// TwinCAT 3 PLC project Lectures
// ProgramVersion: 3.1.4024.0
// libraries:
//   Tc2_Standard, * (Beckhoff Automation GmbH)
//   Tc2_System, * (Beckhoff Automation GmbH)
//   Tc3_Module, * (Beckhoff Automation GmbH)
// project tree:
//   DUTs/ Item.TcDUT (not stored), Location.TcDUT (not stored)
//   GVLs/ Automatic.TcGVL, IO.TcGVL
//   / PlcTask.TcTTO (not stored)
//   POUs/ AutomaticControl.TcPOU, CountPosition.TcPOU (not stored), Initialize.TcPOU, ManualControl.TcPOU, MAIN.TcPOU, MotorSelection.TcPOU, Recipe1.TcPOU, Recipe2.TcPOU, Safety.TcPOU
//   POUs/Lectures%27 programs/ p00_true_false.TcPOU (not stored), p01_sequential.TcPOU (not stored), p02_clock.TcPOU (not stored), p03_SR1.TcPOU (not stored), p04_latch.TcPOU (not stored), p05_posEdge.TcPOU (not stored), p06_frontDetection.TcPOU (not stored), p07_memoryCell.TcPOU (not stored), p08_counter.TcPOU (not stored), p09_timers.TcPOU (not stored), p10_directionalInterlock.TcPOU (not stored), p11_logicalFunction.TcPOU (not stored), p12_controlLight.TcPOU (not stored)
// real-time tasks:
//   TASK PlcTask1: cycle T#10ms, priority 21, ADS port 351
//   TASK PlcTask: cycle T#10ms, priority 20, ADS port 350
// I/O:
//   DEVICE Device 1 (EtherCAT), AmsNetId 172.31.192.1.2.1
//     Term 1 (EK1200) [EK1200-7000 EtherCAT Power supply (1,5A E-Bus)]
//       Term 2 (EL1859) [EL1859 8Ch. Dig. Input 24V, 3ms, 8Ch. Dig. Output 24V, 0.5A]
//       Term 3 (EL1859) [EL1859 8Ch. Dig. Input 24V, 3ms, 8Ch. Dig. Output 24V, 0.5A]
//       Term 4 (EL9011) [EL9011 End Terminal]
//   DEVICE Device 2 (NOV-DP-RAM) (disabled)
//   DEVICE Device 3 (CX7000), AmsNetId 172.31.192.1.4.1
//     Term 1 (CX7028) [CX7028-0000-0121]
//       modules: Module 1 (DIO_2x), Module 2 (Empty Module), Module 3 (DIO_2x), Module 4 (Empty Module), Module 5 (DI_2x), Module 6 (Empty Module), Module 7 (DI_2x), Module 8 (Empty Module)
// variable links:
//   Lectures/Lectures Instance <-> Device 1 (EtherCAT)/Term 1 (EK1200)/Term 2 (EL1859)
//     PlcTask Inputs/IO.EndExtensionSensor <-> Channel 3/Input
//     PlcTask Inputs/IO.EndGripSensor <-> Channel 7/Input
//     PlcTask Inputs/IO.EndLiftingSensor <-> Channel 5/Input
//     PlcTask Inputs/IO.EndRotationSensor <-> Channel 1/Input
//     PlcTask Inputs/IO.StepExtensionSwitch <-> Channel 4/Input
//     PlcTask Inputs/IO.StepGripSwitch <-> Channel 8/Input
//     PlcTask Inputs/IO.StepLiftingSwitch <-> Channel 6/Input
//     PlcTask Inputs/IO.StepRotatonSwitch <-> Channel 2/Input
//     PlcTask Outputs/IO.MotorExtension <-> Channel 12/Output
//     PlcTask Outputs/IO.MotorExtensionDirection <-> Channel 11/Output
//     PlcTask Outputs/IO.MotorGrip <-> Channel 16/Output
//     PlcTask Outputs/IO.MotorGripDirection <-> Channel 15/Output
//     PlcTask Outputs/IO.MotorLifting <-> Channel 14/Output
//     PlcTask Outputs/IO.MotorLiftingDirection <-> Channel 13/Output
//     PlcTask Outputs/IO.MotorRotation <-> Channel 10/Output
//     PlcTask Outputs/IO.MotorRotationDirection <-> Channel 9/Output
//   Lectures/Lectures Instance <-> Device 3 (CX7000)/Term 1 (CX7028)
//     PlcTask Inputs/IO.ButtonGreen <-> Module 3 (DIO_2x)/DIO_2x Input Channel 2/Input
//     PlcTask Inputs/IO.ButtonLowerLeft <-> Module 5 (DI_2x)/DI_2x Input Channel 1/Input
//     PlcTask Inputs/IO.ButtonLowerRight <-> Module 5 (DI_2x)/DI_2x Input Channel 2/Input
//     PlcTask Inputs/IO.ButtonRed <-> Module 1 (DIO_2x)/DIO_2x Input Channel 1/Input
//     PlcTask Inputs/IO.ButtonUpperLeft <-> Module 1 (DIO_2x)/DIO_2x Input Channel 2/Input
//     PlcTask Inputs/IO.ButtonUpperRight <-> Module 3 (DIO_2x)/DIO_2x Input Channel 1/Input
//     PlcTask Inputs/IO.Switch <-> Module 7 (DI_2x)/DI_2x Input Channel 1/Input
//     PlcTask Outputs/IO.LEDBlueLower <-> Module 3 (DIO_2x)/DIO_2x Output Channel 2/Output
//     PlcTask Outputs/IO.LEDBlueUpper <-> Module 1 (DIO_2x)/DIO_2x Output Channel 2/Output
//     PlcTask Outputs/IO.LEDGreen <-> Module 3 (DIO_2x)/DIO_2x Output Channel 1/Output
//     PlcTask Outputs/IO.LEDRed <-> Module 1 (DIO_2x)/DIO_2x Output Channel 1/Output

// ---- GVLs/Automatic.TcGVL
{attribute 'qualified_only'}
VAR_GLOBAL
	SwitchedON: BOOL;
	CurrentLocation: Location;
	CurrentSelection: INT;
	//MotorRot: Motors;
	//MotorLif: Motors;
	//MotorExt: Motors;
	//MotorGri: Motors;
	
	RotationPositionAuto: INT;
	RotationPositionCurrent: INT;
	RotationMovement: BOOL;
	
	LiftingPositionAuto: INT;
	LiftingPositionCurrent: INT;
	LiftingMovement: BOOL;
	
	ExtensionPositionAuto: INT;
	ExtensionPositionCurrent: INT;
	ExtensionMovement: BOOL;
	
	GripPositionAuto: INT;
	GripPositionCurrent: INT;
	GripMovement: BOOL;
END_VAR

// ---- GVLs/IO.TcGVL
{attribute 'qualified_only'}
VAR_GLOBAL
	ButtonRed AT %I*: BOOL;
	ButtonUpperRight AT %I*: BOOL;
	ButtonLowerLeft AT %I*: BOOL;
	Switch AT %I*: BOOL;
	LEDRed AT %Q*: BOOL;
	LEDGreen AT %Q*: BOOL;
	ButtonUpperLeft AT %I*: BOOL;
	ButtonGreen AT %I*: BOOL;
	ButtonLowerRight AT %I*: BOOL;
	LEDBlueUpper AT %Q*: BOOL;
	LEDBlueLower AT %Q*: BOOL;
	
	EndRotationSensor AT %I*: BOOL;
	StepRotatonSwitch AT %I*: BOOL;
	EndExtensionSensor AT %I*: BOOL;
	StepExtensionSwitch AT %I*: BOOL;
	EndLiftingSensor AT %I*: BOOL;
	StepLiftingSwitch AT %I*: BOOL;
	EndGripSensor AT %I*: BOOL;
	StepGripSwitch AT %I*: BOOL;
	MotorRotationDirection AT %Q*: BOOL;
	MotorRotation AT %Q*: BOOL;
	MotorExtensionDirection AT %Q*: BOOL;
	MotorExtension AT %Q*: BOOL;
	MotorLiftingDirection AT %Q*: BOOL;
	MotorLifting AT %Q*: BOOL;
	MotorGripDirection AT %Q*: BOOL;
	MotorGrip AT %Q*: BOOL;
	Initialized: BOOL;
	MotorDirection: INT;
	SwitchedToAutomatic: BOOL;
END_VAR

// ---- POUs/AutomaticControl.TcPOU
FUNCTION_BLOCK PUBLIC AutomaticControl
VAR_INPUT
	Switch: BOOL;
END_VAR
VAR
	ExecutingRecipe1: BOOL := FALSE;
	ExecutingRecipe2: BOOL := FALSE;
	SwitchedManualAuto: BOOL := FALSE;
	initialized: BOOL := FALSE;
	State: INT := 0;
END_VAR
VAR_OUTPUT
	Output: BOOL;
END_VAR

// Initially go to position (0,0,0,0) and initialize motors
IF NOT IO.Initialized THEN
	Initialize();
ELSE
	//Safety();	// to stop when out of range
	
	// COUNTING (POSITION):
	CountPosition();	// FOR MANUAL MODE
	
	// RESET THE POSITION:
	(*IF (Automatic.RotationPositionAuto - Automatic.RotationPositionCurrent > 20 OR Automatic.RotationPositionAuto - Automatic.RotationPositionCurrent > 20) AND IO.SwitchedToAutomatic THEN
		IF Automatic.RotationPositionAuto - Automatic.RotationPositionCurrent > 20 THEN
			IO.MotorRotationDirection := 0;
		ELSE
			IO.MotorRotationDirection := 1;
		END_IF
		IO.MotorRotation := 1;
	ELSE 
		IO.MotorRotation := 0;
		IO.SwitchedToAutomatic := 0;
	END_IF*)
	(*IF Automatic.ExtensionPositionAuto <> Automatic.ExtensionPositionCurrent AND NOT IO.Switch THEN
		IF Automatic.ExtensionPositionAuto - Automatic.ExtensionPositionCurrent > 0 THEN
			IO.MotorExtensionDirection := 0;
		ELSE
			IO.MotorExtensionDirection := 1;
		END_IF
		IO.MotorExtension := 1;
	ELSE 
		IF NOT IO.Switch THEN
			IO.MotorExtension := 0;
		END_IF
	END_IF*)
	
	
	
	// RECIPES (recipe is sequence of moves to execute the task):
	IF ExecutingRecipe1 OR IO.ButtonUpperLeft THEN
		ExecutingRecipe1 := TRUE;
		Recipe1();
		ExecutingRecipe1 := NOT Recipe1.Ended;
	ELSIF NOT ExecutingRecipe1 AND (IO.ButtonUpperRight OR ExecutingRecipe2) THEN
		ExecutingRecipe2 := TRUE;
		Recipe2();
		ExecutingRecipe2 := NOT Recipe2.Ended;
	END_IF
	
END_IF

// for debugging purposes:
IF IO.ButtonRed THEN
	IO.Initialized := FALSE;
END_IF

RETURN;

END_FUNCTION_BLOCK

// ---- POUs/Initialize.TcPOU
PROGRAM Initialize
VAR
END_VAR

// go to the initial position (0,0,0,0)
IF IO.EndRotationSensor THEN
	IO.MotorRotation := 0;
	IO.MotorRotationDirection := 0;
ELSE 
	IO.MotorRotationDirection := 1;
	IO.MotorRotation := 1;
END_IF

IF IO.EndLiftingSensor THEN
	IO.MotorLifting := 0;
	IO.MotorLiftingDirection := 0;
ELSE 
	IO.MotorLiftingDirection := 1;
	IO.MotorLifting := 1;
END_IF

IF IO.EndExtensionSensor THEN
	IO.MotorExtension := 0;
	IO.MotorExtensionDirection := 0;
ELSE 
	IO.MotorExtensionDirection := 1;
	IO.MotorExtension := 1;
END_IF

IF IO.EndGripSensor THEN
	IO.MotorGrip := 0;
	IO.MotorGripDirection := 0;
ELSE 
	IO.MotorGripDirection := 1;
	IO.MotorGrip := 1;
END_IF
	
IF IO.EndRotationSensor AND IO.EndLiftingSensor AND IO.EndExtensionSensor AND IO.EndGripSensor THEN
	IO.Initialized := TRUE;
END_IF

END_PROGRAM

// ---- POUs/Recipe1.TcPOU
PROGRAM Recipe1
VAR
	State: INT := 0;
END_VAR

IF State = 24 AND IO.ButtonGreen THEN	// reinitialize and run the recipe again on green button press
	IO.Initialized := 0;
	State := 0;
END_IF

IF IO.Initialized AND NOT IO.Switch THEN
	
	// delay...
	// vrni se v stanje ob preklopu...
	// daj v funkcije in kliči, namesto PRG...
	// Recipe2...
	
	// WOOD:
	IF State = 0 THEN
		IF Automatic.LiftingPositionAuto < 50 THEN
			IO.MotorLiftingDirection := 0;
			IO.MotorLifting := 1;
			Automatic.LiftingPositionAuto := Automatic.LiftingPositionAuto + 1;
			Automatic.LiftingPositionCurrent := Automatic.LiftingPositionCurrent + 1;
		ELSE
			State := 1;
			IO.MotorLifting := 0;
		END_IF
	ELSIF State = 1 THEN
		IF Automatic.ExtensionPositionAuto < 388 THEN
			IO.MotorExtensionDirection := 0;
			IO.MotorExtension := 1;
			Automatic.ExtensionPositionAuto := Automatic.ExtensionPositionAuto + 1;
			Automatic.ExtensionPositionCurrent := Automatic.ExtensionPositionCurrent + 1;
		ELSE
			State := 2;
			IO.MotorExtension := 0;
		END_IF
	ELSIF State = 2 THEN
		IF Automatic.GripPositionAuto < 160 THEN
			IO.MotorGripDirection := 0;
			IO.MotorGrip := 1;
			Automatic.GripPositionAuto := Automatic.GripPositionAuto + 1;
			Automatic.GripPositionCurrent := Automatic.GripPositionCurrent + 1;
		ELSE
			State := 3;
			IO.MotorGrip := 0;
		END_IF
	ELSIF State = 3 THEN
		IF NOT IO.EndLiftingSensor THEN
			IO.MotorLiftingDirection := 0;
			IO.MotorLifting := 1;
			Automatic.LiftingPositionAuto := Automatic.LiftingPositionAuto - 1;
			Automatic.LiftingPositionCurrent := Automatic.LiftingPositionCurrent - 1;
		ELSE
			State := 4;
			IO.MotorLifting := 0;
		END_IF
	ELSIF State = 4 THEN
		IF Automatic.RotationPositionAuto < 300 THEN
			IO.MotorRotationDirection := 0;
			IO.MotorRotation := 1;
			Automatic.RotationPositionAuto := Automatic.RotationPositionAuto + 1;
			Automatic.RotationPositionCurrent := Automatic.RotationPositionCurrent + 1;
		ELSE
			State := 5;
			IO.MotorRotation := 0;
		END_IF
	ELSIF State = 5 THEN
		IF NOT IO.EndExtensionSensor THEN	// it drops wood in the nearest bin
			IO.MotorExtensionDirection := 1;
			IO.MotorExtension := 1;
			Automatic.ExtensionPositionAuto := Automatic.ExtensionPositionAuto - 1;
			Automatic.ExtensionPositionCurrent := Automatic.ExtensionPositionCurrent - 1;
		ELSE
			State := 6;
			IO.MotorExtension := 0;
		END_IF
	ELSIF State = 6 THEN
		IF NOT IO.EndGripSensor THEN
			IO.MotorGripDirection := 1;
			IO.MotorGrip := 1;
			Automatic.GripPositionAuto := Automatic.GripPositionAuto - 1;
			Automatic.GripPositionCurrent := Automatic.GripPositionCurrent - 1;
		ELSE
			State := 7;
			IO.MotorGrip := 0;
		END_IF
	ELSIF State = 7 THEN
		IF NOT IO.EndRotationSensor THEN
			IO.MotorRotationDirection := 1;
			IO.MotorRotation := 1;
			Automatic.RotationPositionAuto := Automatic.RotationPositionAuto - 1;
			Automatic.RotationPositionCurrent := Automatic.RotationPositionCurrent - 1;
		ELSE
			State := 8;
			IO.MotorRotation := 0;
		END_IF
	END_IF
	
	// PLASTICS:
	IF State = 8 THEN
		IF Automatic.LiftingPositionAuto < 250 THEN
			IO.MotorLiftingDirection := 0;
			IO.MotorLifting := 1;
			Automatic.LiftingPositionAuto := Automatic.LiftingPositionAuto + 1;
			Automatic.LiftingPositionCurrent := Automatic.LiftingPositionCurrent + 1;
		ELSE
			State := 9;
			IO.MotorLifting := 0;
		END_IF
	ELSIF State = 9 THEN
		IF Automatic.ExtensionPositionAuto < 388 THEN
			IO.MotorExtensionDirection := 0;
			IO.MotorExtension := 1;
			Automatic.ExtensionPositionAuto := Automatic.ExtensionPositionAuto + 1;
			Automatic.ExtensionPositionCurrent := Automatic.ExtensionPositionCurrent + 1;
		ELSE
			State := 10;
			IO.MotorExtension := 0;
		END_IF
	ELSIF State = 10 THEN
		IF Automatic.GripPositionAuto < 160 THEN
			IO.MotorGripDirection := 0;
			IO.MotorGrip := 1;
			Automatic.GripPositionAuto := Automatic.GripPositionAuto + 1;
			Automatic.GripPositionCurrent := Automatic.GripPositionCurrent + 1;
		ELSE
			State := 11;
			IO.MotorGrip := 0;
		END_IF
	ELSIF State = 11 THEN
		IF NOT IO.EndLiftingSensor THEN
			IO.MotorLiftingDirection := 1;
			IO.MotorLifting := 1;
			Automatic.LiftingPositionAuto := Automatic.LiftingPositionAuto - 1;
			Automatic.LiftingPositionCurrent := Automatic.LiftingPositionCurrent - 1;
		ELSE
			State := 12;
			IO.MotorLifting := 0;
		END_IF
	ELSIF State = 12 THEN
		IF Automatic.RotationPositionAuto < 300 THEN
			IO.MotorRotationDirection := 0;
			IO.MotorRotation := 1;
			Automatic.RotationPositionAuto := Automatic.RotationPositionAuto + 1;
			Automatic.RotationPositionCurrent := Automatic.RotationPositionCurrent + 1;
		ELSE
			State := 13;
			IO.MotorRotation := 0;
		END_IF
	ELSIF State = 13 THEN
		IF Automatic.ExtensionPositionAuto > 300 THEN	// it drops plastics into second nearest bin
			IO.MotorExtensionDirection := 1;
			IO.MotorExtension := 1;
			Automatic.ExtensionPositionAuto := Automatic.ExtensionPositionAuto - 1;
			Automatic.ExtensionPositionCurrent := Automatic.ExtensionPositionCurrent - 1;
		ELSE
			State := 14;
			IO.MotorExtensionDirection := 0;
			IO.MotorExtension := 0;
		END_IF
	ELSIF State = 14 THEN
		IF NOT IO.EndGripSensor THEN
			IO.MotorGripDirection := 1;
			IO.MotorGrip := 1;
			Automatic.GripPositionAuto := Automatic.GripPositionAuto - 1;
			Automatic.GripPositionCurrent := Automatic.GripPositionCurrent - 1;
		ELSE
			State := 15;
			IO.MotorGrip := 0;
		END_IF
	ELSIF State = 15 THEN
		IF NOT IO.EndRotationSensor THEN
			IO.MotorRotationDirection := 1;
			IO.MotorRotation := 1;
			Automatic.RotationPositionAuto := Automatic.RotationPositionAuto - 1;
			Automatic.RotationPositionCurrent := Automatic.RotationPositionCurrent - 1;
		ELSE
			State := 16;
			IO.MotorRotation := 0;
		END_IF
	END_IF
	
	// METAL:
	IF State = 16 THEN
		IF Automatic.LiftingPositionAuto < 400 THEN
			IO.MotorLiftingDirection := 0;
			IO.MotorLifting := 1;
			Automatic.LiftingPositionAuto := Automatic.LiftingPositionAuto + 1;
			Automatic.LiftingPositionCurrent := Automatic.LiftingPositionCurrent + 1;
		ELSE
			State := 17;
			IO.MotorLifting := 0;
		END_IF
	ELSIF State = 17 THEN
		IF Automatic.ExtensionPositionAuto < 388 THEN
			IO.MotorExtensionDirection := 0;
			IO.MotorExtension := 1;
			Automatic.ExtensionPositionAuto := Automatic.ExtensionPositionAuto + 1;
			Automatic.ExtensionPositionCurrent := Automatic.ExtensionPositionCurrent + 1;
		ELSE
			State := 18;
			IO.MotorExtension := 0;
		END_IF
	ELSIF State = 18 THEN
		IF Automatic.GripPositionAuto < 160 THEN
			IO.MotorGripDirection := 0;
			IO.MotorGrip := 1;
			Automatic.GripPositionAuto := Automatic.GripPositionAuto + 1;
			Automatic.GripPositionCurrent := Automatic.GripPositionCurrent + 1;
		ELSE
			State := 19;
			IO.MotorGrip := 0;
		END_IF
	ELSIF State = 19 THEN
		IF NOT IO.EndLiftingSensor THEN
			IO.MotorLiftingDirection := 1;
			IO.MotorLifting := 1;
			Automatic.LiftingPositionAuto := Automatic.LiftingPositionAuto - 1;
			Automatic.LiftingPositionCurrent := Automatic.LiftingPositionCurrent - 1;
		ELSE
			State := 20;
			IO.MotorLifting := 0;
		END_IF
	ELSIF State = 20 THEN
		IF Automatic.RotationPositionAuto < 300 THEN
			IO.MotorRotationDirection := 0;
			IO.MotorRotation := 1;
			Automatic.RotationPositionAuto := Automatic.RotationPositionAuto + 1;
			Automatic.RotationPositionCurrent := Automatic.RotationPositionCurrent + 1;
		ELSE
			State := 21;
			IO.MotorRotation := 0;
		END_IF
	ELSIF State = 21 THEN
		IF Automatic.ExtensionPositionAuto > 500 THEN	// it drops metal into farthest bin
			IO.MotorExtensionDirection := 1;
			IO.MotorExtension := 1;
			Automatic.ExtensionPositionAuto := Automatic.ExtensionPositionAuto - 1;
			Automatic.ExtensionPositionCurrent := Automatic.ExtensionPositionCurrent - 1;
		ELSE
			State := 22;
			IO.MotorExtension := 0;
		END_IF
	ELSIF State = 22 THEN
		IF NOT IO.EndGripSensor THEN
			IO.MotorGripDirection := 1;
			IO.MotorGrip := 1;
			Automatic.GripPositionAuto := Automatic.GripPositionAuto - 1;
			Automatic.GripPositionCurrent := Automatic.GripPositionCurrent - 1;
		ELSE
			State := 23;
			IO.MotorGrip := 0;
		END_IF
	ELSIF State = 23 THEN
		IF NOT IO.EndRotationSensor THEN
			IO.MotorRotationDirection := 1;
			IO.MotorRotation := 1;
			Automatic.RotationPositionAuto := Automatic.RotationPositionAuto - 1;
			Automatic.RotationPositionCurrent := Automatic.RotationPositionCurrent - 1;
		ELSE
			State := 24;
			IO.MotorRotation := 0;
		END_IF
	END_IF
END_IF

END_PROGRAM

// ---- POUs/Recipe2.TcPOU
PROGRAM Recipe2
VAR
	State: INT := 8;
	Ended: BOOL := FALSE;
END_VAR

IF State = 24 AND IO.ButtonGreen THEN	// reinitialize and run the recipe again on green button press
	IO.Initialized := 0;
	State := 0;
END_IF

IF IO.Initialized AND NOT IO.Switch THEN
	
	// WOOD:
	IF State = 0 THEN
		IF Automatic.LiftingPositionAuto < 50 THEN
			IO.MotorLiftingDirection := 0;
			IO.MotorLifting := 1;
			Automatic.LiftingPositionAuto := Automatic.LiftingPositionAuto + 1;
			Automatic.LiftingPositionCurrent := Automatic.LiftingPositionCurrent + 1;
		ELSE
			State := 1;
			IO.MotorLifting := 0;
		END_IF
	ELSIF State = 1 THEN
		IF Automatic.ExtensionPositionAuto < 388 THEN
			IO.MotorExtensionDirection := 0;
			IO.MotorExtension := 1;
			Automatic.ExtensionPositionAuto := Automatic.ExtensionPositionAuto + 1;
			Automatic.ExtensionPositionCurrent := Automatic.ExtensionPositionCurrent + 1;
		ELSE
			State := 2;
			IO.MotorExtension := 0;
		END_IF
	ELSIF State = 2 THEN
		IF Automatic.GripPositionAuto < 160 THEN
			IO.MotorGripDirection := 0;
			IO.MotorGrip := 1;
			Automatic.GripPositionAuto := Automatic.GripPositionAuto + 1;
			Automatic.GripPositionCurrent := Automatic.GripPositionCurrent + 1;
		ELSE
			State := 3;
			IO.MotorGrip := 0;
		END_IF
	ELSIF State = 3 THEN
		IF NOT IO.EndLiftingSensor THEN
			IO.MotorLiftingDirection := 1;
			IO.MotorLifting := 1;
			Automatic.LiftingPositionAuto := Automatic.LiftingPositionAuto - 1;
			Automatic.LiftingPositionCurrent := Automatic.LiftingPositionCurrent - 1;
		ELSE
			State := 4;
			IO.MotorLifting := 0;
		END_IF
	ELSIF State = 4 THEN
		IF Automatic.RotationPositionAuto < 300 THEN
			IO.MotorRotationDirection := 0;
			IO.MotorRotation := 1;
			Automatic.RotationPositionAuto := Automatic.RotationPositionAuto + 1;
			Automatic.RotationPositionCurrent := Automatic.RotationPositionCurrent + 1;
		ELSE
			State := 5;
			IO.MotorRotation := 0;
		END_IF
	ELSIF State = 5 THEN
		IF NOT IO.EndExtensionSensor THEN	// it drops wood in the nearest bin
			IO.MotorExtensionDirection := 1;
			IO.MotorExtension := 1;
			Automatic.ExtensionPositionAuto := Automatic.ExtensionPositionAuto - 1;
			Automatic.ExtensionPositionCurrent := Automatic.ExtensionPositionCurrent - 1;
		ELSE
			State := 6;
			IO.MotorExtension := 0;
		END_IF
	ELSIF State = 6 THEN
		IF NOT IO.EndGripSensor THEN
			IO.MotorGripDirection := 1;
			IO.MotorGrip := 1;
			Automatic.GripPositionAuto := Automatic.GripPositionAuto - 1;
			Automatic.GripPositionCurrent := Automatic.GripPositionCurrent - 1;
		ELSE
			State := 7;
			IO.MotorGrip := 0;
		END_IF
	ELSIF State = 7 THEN
		IF NOT IO.EndRotationSensor THEN
			IO.MotorRotationDirection := 1;
			IO.MotorRotation := 1;
			Automatic.RotationPositionAuto := Automatic.RotationPositionAuto - 1;
			Automatic.RotationPositionCurrent := Automatic.RotationPositionCurrent - 1;
		ELSE
			State := 8;
			IO.MotorRotation := 0;
		END_IF
	END_IF
	
	// PLASTICS:
	IF State = 8 THEN
		IF Automatic.LiftingPositionAuto < 250 THEN
			IO.MotorLiftingDirection := 0;
			IO.MotorLifting := 1;
			Automatic.LiftingPositionAuto := Automatic.LiftingPositionAuto + 1;
			Automatic.LiftingPositionCurrent := Automatic.LiftingPositionCurrent + 1;
		ELSE
			State := 9;
			IO.MotorLifting := 0;
		END_IF
	ELSIF State = 9 THEN
		IF Automatic.ExtensionPositionAuto < 388 THEN
			IO.MotorExtensionDirection := 0;
			IO.MotorExtension := 1;
			Automatic.ExtensionPositionAuto := Automatic.ExtensionPositionAuto + 1;
			Automatic.ExtensionPositionCurrent := Automatic.ExtensionPositionCurrent + 1;
		ELSE
			State := 10;
			IO.MotorExtension := 0;
		END_IF
	ELSIF State = 10 THEN
		IF Automatic.GripPositionAuto < 160 THEN
			IO.MotorGripDirection := 0;
			IO.MotorGrip := 1;
			Automatic.GripPositionAuto := Automatic.GripPositionAuto + 1;
			Automatic.GripPositionCurrent := Automatic.GripPositionCurrent + 1;
		ELSE
			State := 11;
			IO.MotorGrip := 0;
		END_IF
	ELSIF State = 11 THEN
		IF NOT IO.EndLiftingSensor THEN
			IO.MotorLiftingDirection := 1;
			IO.MotorLifting := 1;
			Automatic.LiftingPositionAuto := Automatic.LiftingPositionAuto - 1;
			Automatic.LiftingPositionCurrent := Automatic.LiftingPositionCurrent - 1;
		ELSE
			State := 12;
			IO.MotorLifting := 0;
		END_IF
	ELSIF State = 12 THEN
		IF Automatic.RotationPositionAuto < 300 THEN
			IO.MotorRotationDirection := 0;
			IO.MotorRotation := 1;
			Automatic.RotationPositionAuto := Automatic.RotationPositionAuto + 1;
			Automatic.RotationPositionCurrent := Automatic.RotationPositionCurrent + 1;
		ELSE
			State := 13;
			IO.MotorRotation := 0;
		END_IF
	ELSIF State = 13 THEN
		IF Automatic.ExtensionPositionAuto > 300 THEN	// it drops plastics into second nearest bin
			IO.MotorExtensionDirection := 1;
			IO.MotorExtension := 1;
			Automatic.ExtensionPositionAuto := Automatic.ExtensionPositionAuto - 1;
			Automatic.ExtensionPositionCurrent := Automatic.ExtensionPositionCurrent - 1;
		ELSE
			State := 14;
			IO.MotorExtensionDirection := 0;
			IO.MotorExtension := 0;
		END_IF
	ELSIF State = 14 THEN
		IF NOT IO.EndGripSensor THEN
			IO.MotorGripDirection := 1;
			IO.MotorGrip := 1;
			Automatic.GripPositionAuto := Automatic.GripPositionAuto - 1;
			Automatic.GripPositionCurrent := Automatic.GripPositionCurrent - 1;
		ELSE
			State := 15;
			IO.MotorGrip := 0;
		END_IF
	ELSIF State = 15 THEN
		IF NOT IO.EndRotationSensor THEN
			IO.MotorRotationDirection := 1;
			IO.MotorRotation := 1;
			Automatic.RotationPositionAuto := Automatic.RotationPositionAuto - 1;
			Automatic.RotationPositionCurrent := Automatic.RotationPositionCurrent - 1;
		ELSE
			State := 16;
			IO.MotorRotation := 0;
		END_IF
	END_IF
	
	// METAL:
	IF State = 16 THEN
		IF Automatic.LiftingPositionAuto < 400 THEN
			IO.MotorLiftingDirection := 0;
			IO.MotorLifting := 1;
			Automatic.LiftingPositionAuto := Automatic.LiftingPositionAuto + 1;
			Automatic.LiftingPositionCurrent := Automatic.LiftingPositionCurrent + 1;
		ELSE
			State := 17;
			IO.MotorLifting := 0;
		END_IF
	ELSIF State = 17 THEN
		IF Automatic.ExtensionPositionAuto < 388 THEN
			IO.MotorExtensionDirection := 0;
			IO.MotorExtension := 1;
			Automatic.ExtensionPositionAuto := Automatic.ExtensionPositionAuto + 1;
			Automatic.ExtensionPositionCurrent := Automatic.ExtensionPositionCurrent + 1;
		ELSE
			State := 18;
			IO.MotorExtension := 0;
		END_IF
	ELSIF State = 18 THEN
		IF Automatic.GripPositionAuto < 160 THEN
			IO.MotorGripDirection := 0;
			IO.MotorGrip := 1;
			Automatic.GripPositionAuto := Automatic.GripPositionAuto + 1;
			Automatic.GripPositionCurrent := Automatic.GripPositionCurrent + 1;
		ELSE
			State := 19;
			IO.MotorGrip := 0;
		END_IF
	ELSIF State = 19 THEN
		IF NOT IO.EndLiftingSensor THEN
			IO.MotorLiftingDirection := 1;
			IO.MotorLifting := 1;
			Automatic.LiftingPositionAuto := Automatic.LiftingPositionAuto - 1;
			Automatic.LiftingPositionCurrent := Automatic.LiftingPositionCurrent - 1;
		ELSE
			State := 20;
			IO.MotorLifting := 0;
		END_IF
	ELSIF State = 20 THEN
		IF Automatic.RotationPositionAuto < 300 THEN
			IO.MotorRotationDirection := 0;
			IO.MotorRotation := 1;
			Automatic.RotationPositionAuto := Automatic.RotationPositionAuto + 1;
			Automatic.RotationPositionCurrent := Automatic.RotationPositionCurrent + 1;
		ELSE
			State := 21;
			IO.MotorRotation := 0;
		END_IF
	ELSIF State = 21 THEN
		IF Automatic.ExtensionPositionAuto > 500 THEN	// it drops metal into farthest bin
			IO.MotorExtensionDirection := 1;
			IO.MotorExtension := 1;
			Automatic.ExtensionPositionAuto := Automatic.ExtensionPositionAuto - 1;
			Automatic.ExtensionPositionCurrent := Automatic.ExtensionPositionCurrent - 1;
		ELSE
			State := 22;
			IO.MotorExtension := 0;
		END_IF
	ELSIF State = 22 THEN
		IF NOT IO.EndGripSensor THEN
			IO.MotorGripDirection := 1;
			IO.MotorGrip := 1;
			Automatic.GripPositionAuto := Automatic.GripPositionAuto - 1;
			Automatic.GripPositionCurrent := Automatic.GripPositionCurrent - 1;
		ELSE
			State := 23;
			IO.MotorGrip := 0;
		END_IF
	ELSIF State = 23 THEN
		IF NOT IO.EndRotationSensor THEN
			IO.MotorRotationDirection := 1;
			IO.MotorRotation := 1;
			Automatic.RotationPositionAuto := Automatic.RotationPositionAuto - 1;
			Automatic.RotationPositionCurrent := Automatic.RotationPositionCurrent - 1;
		ELSE
			State := 24;
			IO.MotorRotation := 0;
		END_IF
	ELSIF State = 24 THEN
		State := 8;
		Ended := TRUE;
	END_IF
END_IF

END_PROGRAM

// ---- POUs/ManualControl.TcPOU
FUNCTION_BLOCK PUBLIC ManualControl
VAR_INPUT
	Switch: BOOL;
END_VAR
VAR
	ManualControl: BOOL;
	TimeForInterlockDelay: TIME := T#0.05S;
	ManualMode: BOOL;
	MotorSelection_1: MotorSelection;
	SelectedMotor: INT;
	temp: TIME;
	LowerLeftInterlock: TOF;
	LowerLeft: BOOL;
	LowerRightInterlock: TOF;
	LowerRight: BOOL;
END_VAR
VAR_OUTPUT
	Output: BOOL;
END_VAR
VAR // added by the converter: edge detectors and wires of the graphical bodies
    _w1, _w2, _w3, _w4, _w5 : BOOL;
END_VAR

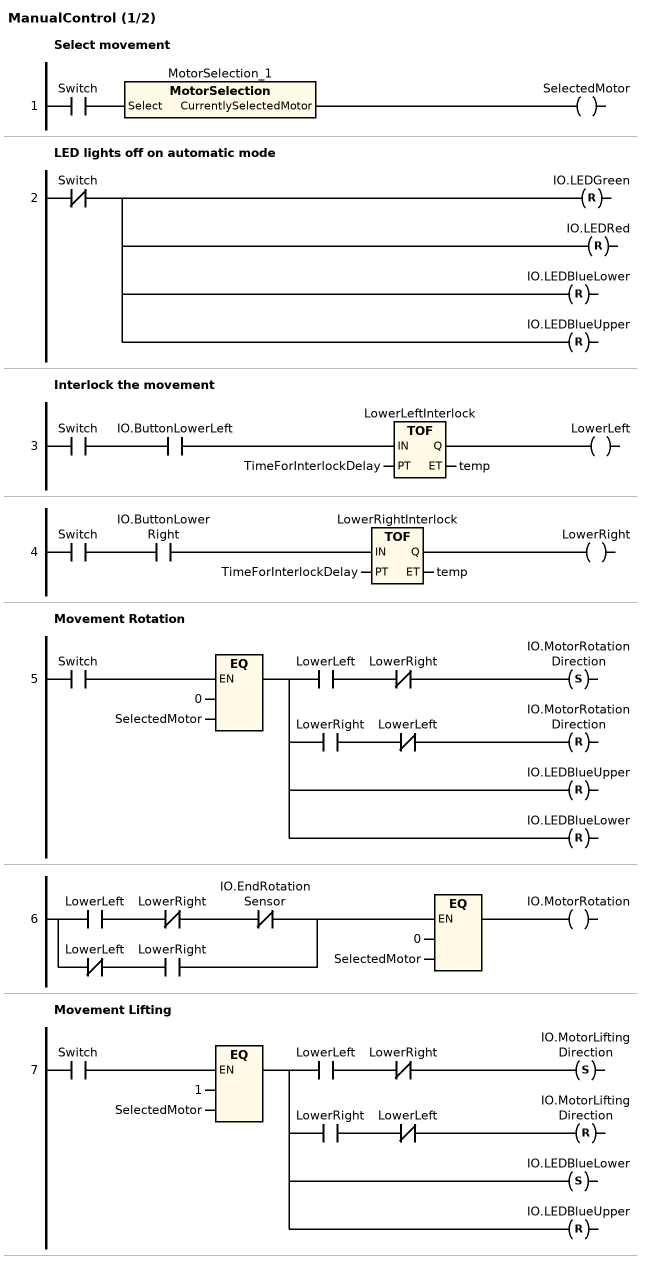
// NETWORK 1: Select movement
MotorSelection_1(Select := Switch); // MotorSelection
SelectedMotor := MotorSelection_1.CurrentlySelectedMotor;

// NETWORK 2: LED lights off on automatic mode
_w1 := NOT Switch;
IO.LEDGreen R= _w1;
IO.LEDRed R= _w1;
IO.LEDBlueLower R= _w1;
IO.LEDBlueUpper R= _w1;

// NETWORK 3: Interlock the movement
LowerLeftInterlock(IN := Switch AND IO.ButtonLowerLeft, PT := TimeForInterlockDelay, ET => temp); // TOF
LowerLeft := LowerLeftInterlock.Q;

// NETWORK 4
LowerRightInterlock(IN := Switch AND IO.ButtonLowerRight, PT := TimeForInterlockDelay, ET => temp); // TOF
LowerRight := LowerRightInterlock.Q;

// NETWORK 5: Movement Rotation
_w2 := Switch AND 0 = SelectedMotor;
IO.MotorRotationDirection S= _w2 AND LowerLeft AND NOT LowerRight;
IO.MotorRotationDirection R= _w2 AND LowerRight AND NOT LowerLeft;
IO.LEDBlueUpper R= _w2;
IO.LEDBlueLower R= _w2;

// NETWORK 6
IO.MotorRotation := (LowerLeft AND NOT LowerRight AND NOT IO.EndRotationSensor OR NOT LowerLeft AND LowerRight) AND 0 = SelectedMotor;

// NETWORK 7: Movement Lifting
_w3 := Switch AND 1 = SelectedMotor;
IO.MotorLiftingDirection S= _w3 AND LowerLeft AND NOT LowerRight;
IO.MotorLiftingDirection R= _w3 AND LowerRight AND NOT LowerLeft;
IO.LEDBlueLower S= _w3;
IO.LEDBlueUpper R= _w3;

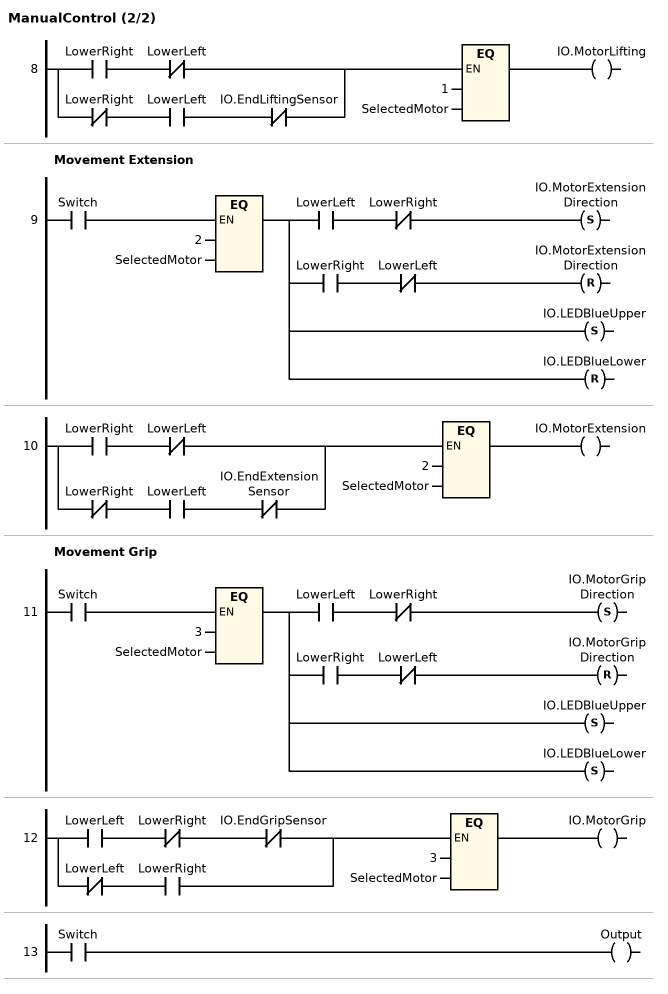
// NETWORK 8
IO.MotorLifting := (LowerRight AND NOT LowerLeft OR NOT LowerRight AND LowerLeft AND NOT IO.EndLiftingSensor) AND 1 = SelectedMotor;

// NETWORK 9: Movement Extension
_w4 := Switch AND 2 = SelectedMotor;
IO.MotorExtensionDirection S= _w4 AND LowerLeft AND NOT LowerRight;
IO.MotorExtensionDirection R= _w4 AND LowerRight AND NOT LowerLeft;
IO.LEDBlueUpper S= _w4;
IO.LEDBlueLower R= _w4;

// NETWORK 10
IO.MotorExtension := (LowerRight AND NOT LowerLeft OR NOT LowerRight AND LowerLeft AND NOT IO.EndExtensionSensor) AND 2 = SelectedMotor;

// NETWORK 11: Movement Grip
_w5 := Switch AND 3 = SelectedMotor;
IO.MotorGripDirection S= _w5 AND LowerLeft AND NOT LowerRight;
IO.MotorGripDirection R= _w5 AND LowerRight AND NOT LowerLeft;
IO.LEDBlueUpper S= _w5;
IO.LEDBlueLower S= _w5;

// NETWORK 12
IO.MotorGrip := (LowerLeft AND NOT LowerRight AND NOT IO.EndGripSensor OR NOT LowerLeft AND LowerRight) AND 3 = SelectedMotor;

// NETWORK 13
Output := Switch;

END_FUNCTION_BLOCK

// ---- POUs/MotorSelection.TcPOU
FUNCTION_BLOCK PUBLIC MotorSelection
VAR_INPUT
	ManualMode: BOOL;
END_VAR
VAR
	TimeForDelay: TIME := T#0.15S;
	MovementSelection: CTUD;
	SelectionCounter: CTUD := (LOAD := TRUE, PV := 3);
	ReachedMaxSelection: BOOL;
	ReachedMinSelection: BOOL;
	UpperLeftDelay: TOF;
	UpperRightDelay: TOF;
	tmnp: TIME;
	CU: BOOL;
	CD: BOOL;
	CUU: BOOL;
	CDD: BOOL;
	PositiveEdge1: R_TRIG;
	PositiveEdge2: R_TRIG;
	temporary: BOOL;
	CUU0: BOOL;
	CDD0: BOOL;
	temporary1: BOOL;
	BURpositiveEdge: BOOL;
	BULpositiveEdge: BOOL;
	temp2: BOOL;
	temp3: BOOL;
END_VAR
VAR_OUTPUT
	CurrentSelection: INT;
END_VAR
VAR // added by the converter: edge detectors and wires of the graphical bodies
    _rt1, _rt2, _rt3, _rt4 : R_TRIG;
END_VAR

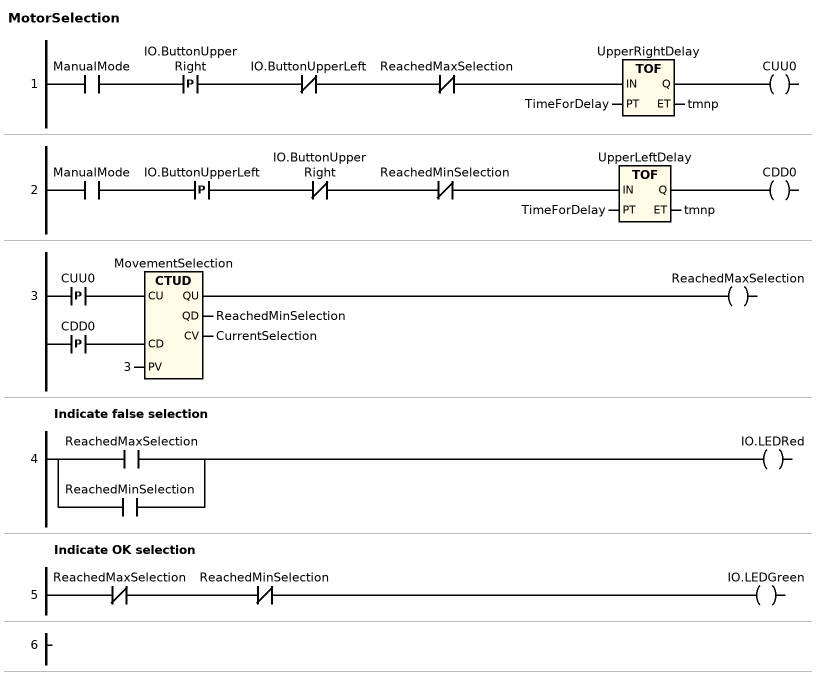
// NETWORK 1
_rt1(CLK := IO.ButtonUpperRight);
UpperRightDelay(
    IN := ManualMode AND _rt1.Q AND NOT IO.ButtonUpperLeft AND NOT ReachedMaxSelection,
    PT := TimeForDelay,
    ET => tmnp); // TOF
CUU0 := UpperRightDelay.Q;

// NETWORK 2
_rt2(CLK := IO.ButtonUpperLeft);
UpperLeftDelay(
    IN := ManualMode AND _rt2.Q AND NOT IO.ButtonUpperRight AND NOT ReachedMinSelection,
    PT := TimeForDelay,
    ET => tmnp); // TOF
CDD0 := UpperLeftDelay.Q;

// NETWORK 3
_rt3(CLK := CUU0);
_rt4(CLK := CDD0);
MovementSelection(CU := _rt3.Q, CD := _rt4.Q, PV := 3, QD => ReachedMinSelection, CV => CurrentSelection); // CTUD
ReachedMaxSelection := MovementSelection.QU;

// NETWORK 4: Indicate false selection
IO.LEDRed := ReachedMaxSelection OR ReachedMinSelection;

// NETWORK 5: Indicate OK selection
IO.LEDGreen := NOT ReachedMaxSelection AND NOT ReachedMinSelection;

// NETWORK 6

END_FUNCTION_BLOCK

// ---- POUs/MAIN.TcPOU
PROGRAM MAIN
VAR
	ManualControl_0: ManualControl;
	AutomaticControl_0: AutomaticControl;
END_VAR

//Functions should ideally avoid changing global or external variables, though this is technically allowed in some cases.
VAR // added by the converter: edge detectors and wires of the graphical bodies
    _w1 : BOOL;
    _rt1 : R_TRIG;
END_VAR

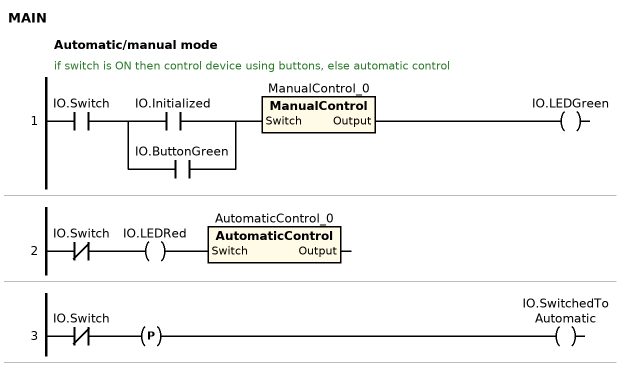
// NETWORK 1: Automatic/manual mode
// if switch is ON then control device using buttons, else automatic control
ManualControl_0(Switch := IO.Switch AND IO.Initialized OR IO.Switch AND IO.ButtonGreen); // ManualControl
IO.LEDGreen := ManualControl_0.Output;

// NETWORK 2
_w1 := NOT IO.Switch;
IO.LEDRed := _w1;
AutomaticControl_0(Switch := _w1); // AutomaticControl

// NETWORK 3
_rt1(CLK := NOT IO.Switch);
IO.SwitchedToAutomatic := _rt1.Q;

END_PROGRAM

// ---- POUs/Safety.TcPOU
PROGRAM Safety
VAR
END_VAR

// Safety for Rotation:
IF Automatic.RotationPositionCurrent >= 570 AND NOT IO.ButtonLowerLeft THEN
	//IO.MotorRotation := 0;
END_IF
IF IO.EndRotationSensor THEN
	Automatic.RotationPositionCurrent := 0;
END_IF

// Safety for Lifting:
IF Automatic.LiftingPositionCurrent >= 355 AND NOT IO.ButtonLowerLeft THEN
	//IO.MotorLifting := 0;
END_IF
IF IO.EndLiftingSensor THEN
	Automatic.LiftingPositionCurrent := 0;
END_IF

// Safety for Extension:
IF Automatic.ExtensionPositionCurrent >= 445 AND NOT IO.ButtonLowerLeft THEN
	//IO.MotorExtension := 0;
END_IF
IF IO.EndExtensionSensor THEN
	Automatic.ExtensionPositionCurrent := 0;
END_IF

// Safety for Grip:
IF Automatic.GripPositionCurrent >= 80 AND NOT IO.ButtonLowerLeft THEN
	//IO.MotorGrip := 0;
END_IF
IF IO.EndGripSensor THEN
	Automatic.GripPositionCurrent := 0;
END_IF

END_PROGRAM
